// TIA Portal V17 export
BLOCK "FC_Jump"   // ObjectSW16, LAD
BEGIN

REGION Network 1: jump label return
END_REGION
END_BLOCK
